TEXTLIST M1ConfigTabsTextList
  0 = 'General'
  1 = 'Radial - General'
  2 = 'Radial - Pressure @ regulator'
  3 = 'Radial - Pressure @ mirror cell'
  4 = 'Axial - General'
  5 = 'Axial - Pressure @ regulator'
  6 = 'Axial - Pressure @ mirror cell'
  7 = 'Axial - Force sensors'
  8 = 'Axial - Average force'
  9 = 'Inclinometer - voltage'
   = ''
END_TEXTLIST

(* stored: Version 1.1.0.1, ProductVersion 3.1.4018.2
   TextList M1ConfigTabsTextList: Id {1ccb876d-33c5-4465-b5a1-09c6bf823c11} *)
